INTERFACE I_EventPublisher EXTENDS I_Observable

PROPERTY Event : int
GET
END_GET
END_PROPERTY

END_INTERFACE

(* stored: Version 1.1.0.1, ProductVersion 3.1.4024.11
   Itf I_EventPublisher: Id {1f5de49e-15f1-4016-8ec5-881bbd6dbdff}
   Property Event: Id {b96138b9-a9e5-4d6c-a65d-f57b15e0a398}
   Get Get: Id {f8cdae7e-232d-4e5e-a739-7f4256dc9b12} *)
